FUNCTION_BLOCK AOI_HeatBase
VAR_INPUT
	Enable: BOOL;
	Reset: BOOL;
	PV: REAL;
	SV: REAL;
	HighLimit: REAL;
	LowLimit: REAL;
	MaxLimit: REAL;
	Kp: REAL:=0.8;
	Ki: REAL:=1;
	Kd: REAL:=5;
END_VAR
VAR_OUTPUT
	Active: BOOL;
	Error: BOOL;
	ErrorID: INT;	
END_VAR
VAR
    blinkAct: blink;
	tonLow: Ton;
	tonHigh: Ton;	
	iDiff: INT;
	arDiff: ARRAY[0..255] OF REAL;
	i: INT;
	n: INT;
	tonSample: Ton;
	rAverageDiff: REAL;
	rSumDiff: REAL;
	j: INT;
	iAct: INT;
	iPID: INT;
	arM: ARRAY[0..255] OF REAL;

	arPV: ARRAY[0..255] OF REAL;
	Mi: REAL;
	MX:REAL;
	Kc: INT:=8;
END_VAR

(*
IF PV < SV AND NOT ErrorID.0 AND NOT ErrorID.1 THEN
	Active:=TRUE;
ELSE 
	Active:=FALSE;
END_IF	  
*)

tonHigh(IN:=(PV> SV+HighLimit) , PT:= T#3S, Q=> , ET=> );
IF tonHigh.Q THEN
	Error:=TRUE;
	ErrorID.0:=TRUE;
END_IF

IF PV>MaxLimit THEN
	Error:=TRUE;        
	ErrorID.1:=TRUE;		
END_IF       

tonLow(IN:=(PV < SV-Lowlimit) , PT:= T#3S, Q=> , ET=> );
IF tonLow.Q THEN
	Error:=TRUE;     
	ErrorID.2:=TRUE;	  
END_IF

IF Reset THEN
	Error:=FALSE;
	ErrorID:=0;
END_IF

CASE iDiff OF
	0:
	  IF Enable THEN
		  iDiff:=1;
	  END_IF
	1:  
	  IF SV>0 THEN
		  IF PV < SV-SV*0.05 THEN
			 iDiff:=100; 
		  END_IF
		  IF PV > SV-SV*0.05 AND NOT ErrorID.0 AND NOT ErrorID.1 THEN
			 rSumDiff:=0;		  
			 iDiff:=10;
		  END_IF
	  END_IF 
	10:
	  arDiff[i]:=SV-PV;
	  IF ABS(arDiff[i]>SV) THEN
		  arDiff[i]:=0;
	  END_IF
	  rSumDiff:=rSumDiff+arDiff[i];
	  (*
	  IF i = Kc THEN
	     rSumDiff:= 0;
	     FOR j:=0 TO Kc DO
		     rSumDiff:= rSumDiff+ arDiff[j];
			 rAverageDiff:=rSumDiff/Kc;
	     END_FOR
	  END_IF  
	  *)
	  iDiff:=20;
	 
    20: 
      arM[0]:=Kp*arDiff[i];
      arM[1]:= Ki*rSumDiff;
	  IF arM[1]>1900 THEN
		 arM[1]:=1900;
	  END_IF
	  IF arM[1]<-1900 THEN
		 arM[1]:=-1900;
	  END_IF
	  
	  IF i=0 THEN
         arM[2]:=Kd*(arDiff[i]-arDiff[Kc]);
	  ELSE
	     arM[2]:=Kd*(arDiff[i]-arDiff[i-1]);
	  END_IF 
	  arM[2]:=arM[2];

	  arM[3]:= (arM[0]+arM[1]+arM[2])*100;
	  IF ARM[3]>1800 THEN
		 ARM[3]:=1800;
		 ELSE IF ARM[3]<200 THEN
			     ARM[3]:=200;
		      END_IF
	  END_IF	
	  iDiff:=30;
	  
	30:  
	  Active:=TRUE;
	  tonSample(IN:= TRUE, PT:= REAL_TO_TIME(arM[3]), Q=> , ET=> );
	  IF tonSample.Q THEN
		  tonSample(IN:= FALSE, PT:= REAL_TO_TIME(arM[3]), Q=> , ET=> );
		  Active:=FALSE;
		  iDiff:=40;
	  END_IF
	40:
	  Active:=FALSE;
	  tonSample(IN:= TRUE, PT:= REAL_TO_TIME(2000-arM[3]), Q=> , ET=> );
	  IF tonSample.Q THEN
		  tonSample(IN:= FALSE, PT:= REAL_TO_TIME(2000-arM[3]), Q=> , ET=> );
		  Active:=FALSE;
		  iDiff:=50;
	  END_IF

	50:  
	  i:=i+1;
	  IF i>Kc THEN
		  i:=0;  
	  END_IF	   
	  iDiff:=0;
	  
	100: 
		IF PV < SV-SV*0.05 AND NOT ErrorID.0 AND NOT ErrorID.1 THEN
			Active:=TRUE;
		ELSE 
			Active:=FALSE;
			iDiff:=0;
		END_IF	  
	  	 
END_CASE

CASE iAct OF 
	0:iAct:=0;
	
END_CASE

END_FUNCTION_BLOCK

(* stored: Version 1.1.0.1, ProductVersion 3.1.4024.6
   POU AOI_HeatBase: Id {b91647b6-7044-4a11-9382-4d7cb2750de3}, SpecialFunc None *)
